// Mitsubishi GX Works2 project: ラダー図整理160913   PLC: Q03UDV

PROGRAM P1
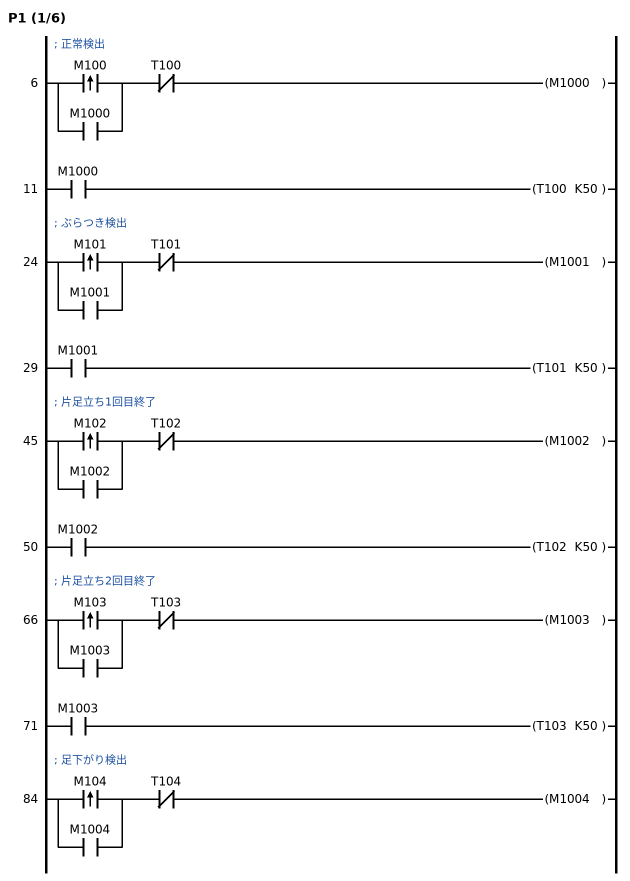
; 正常検出
6     LDP     M100
      OR      M1000
      ANI     T100
      OUT     M1000
11    LD      M1000
      OUT     T100 K50
; ぶらつき検出
24    LDP     M101
      OR      M1001
      ANI     T101
      OUT     M1001
29    LD      M1001
      OUT     T101 K50
; 片足立ち1回目終了
45    LDP     M102
      OR      M1002
      ANI     T102
      OUT     M1002
50    LD      M1002
      OUT     T102 K50
; 片足立ち2回目終了
66    LDP     M103
      OR      M1003
      ANI     T103
      OUT     M1003
71    LD      M1003
      OUT     T103 K50
; 足下がり検出
84    LDP     M104
      OR      M1004
      ANI     T104
      OUT     M1004
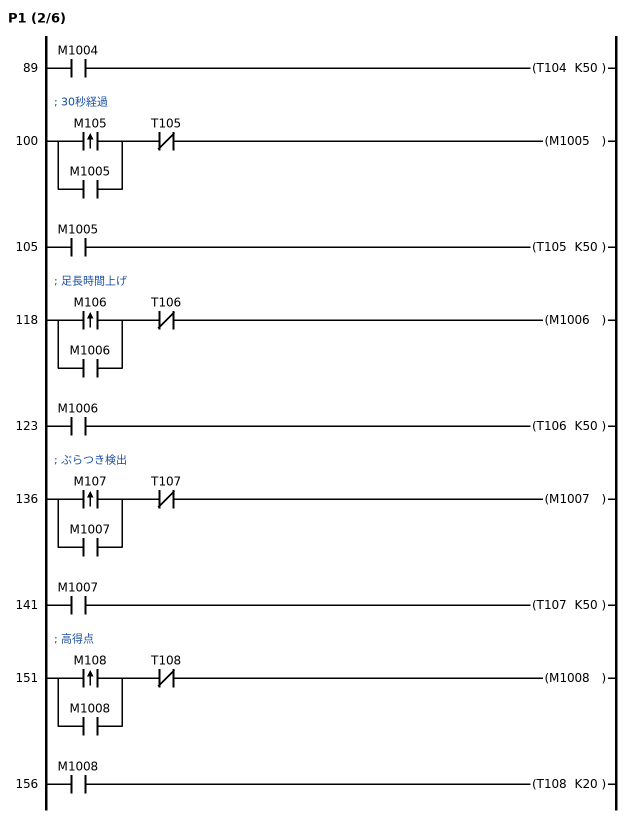
89    LD      M1004
      OUT     T104 K50
; 30秒経過
100   LDP     M105
      OR      M1005
      ANI     T105
      OUT     M1005
105   LD      M1005
      OUT     T105 K50
; 足長時間上げ
118   LDP     M106
      OR      M1006
      ANI     T106
      OUT     M1006
123   LD      M1006
      OUT     T106 K50
; ぶらつき検出
136   LDP     M107
      OR      M1007
      ANI     T107
      OUT     M1007
141   LD      M1007
      OUT     T107 K50
; 高得点
151   LDP     M108
      OR      M1008
      ANI     T108
      OUT     M1008
156   LD      M1008
      OUT     T108 K20
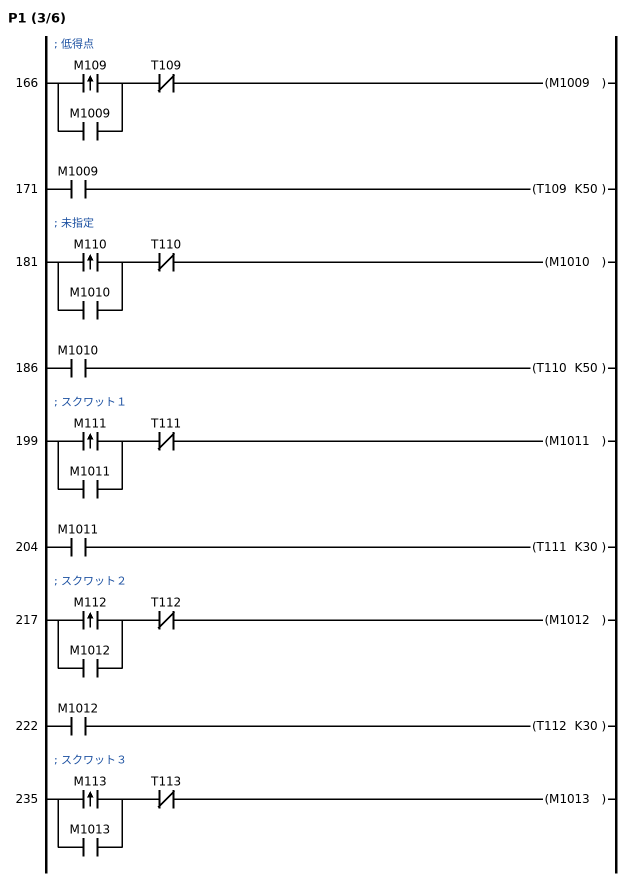
; 低得点
166   LDP     M109
      OR      M1009
      ANI     T109
      OUT     M1009
171   LD      M1009
      OUT     T109 K50
; 未指定
181   LDP     M110
      OR      M1010
      ANI     T110
      OUT     M1010
186   LD      M1010
      OUT     T110 K50
; スクワット１
199   LDP     M111
      OR      M1011
      ANI     T111
      OUT     M1011
204   LD      M1011
      OUT     T111 K30
; スクワット２
217   LDP     M112
      OR      M1012
      ANI     T112
      OUT     M1012
222   LD      M1012
      OUT     T112 K30
; スクワット３
235   LDP     M113
      OR      M1013
      ANI     T113
      OUT     M1013
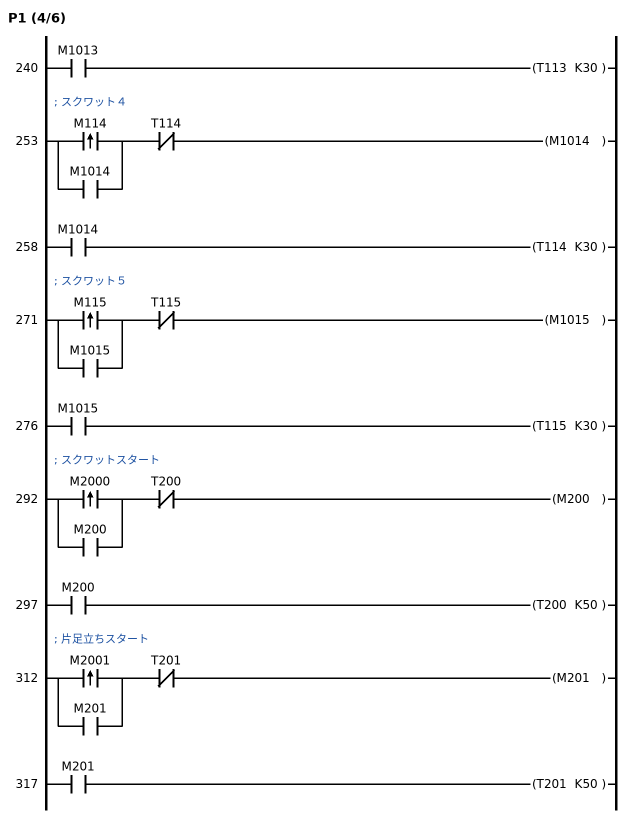
240   LD      M1013
      OUT     T113 K30
; スクワット４
253   LDP     M114
      OR      M1014
      ANI     T114
      OUT     M1014
258   LD      M1014
      OUT     T114 K30
; スクワット５
271   LDP     M115
      OR      M1015
      ANI     T115
      OUT     M1015
276   LD      M1015
      OUT     T115 K30
; スクワットスタート
292   LDP     M2000
      OR      M200
      ANI     T200
      OUT     M200
297   LD      M200
      OUT     T200 K50
; 片足立ちスタート
312   LDP     M2001
      OR      M201
      ANI     T201
      OUT     M201
317   LD      M201
      OUT     T201 K50
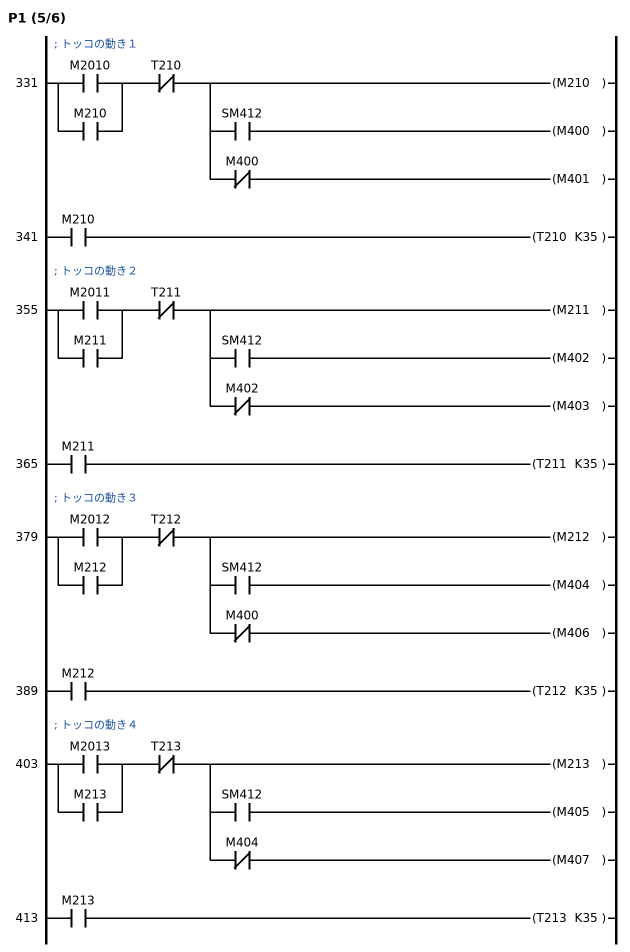
; トッコの動き１
331   LD      M2010
      OR      M210
      ANI     T210
      OUT     M210
      MPS
      AND     SM412
      OUT     M400
      MPP
      ANI     M400
      OUT     M401
341   LD      M210
      OUT     T210 K35
; トッコの動き２
355   LD      M2011
      OR      M211
      ANI     T211
      OUT     M211
      MPS
      AND     SM412
      OUT     M402
      MPP
      ANI     M402
      OUT     M403
365   LD      M211
      OUT     T211 K35
; トッコの動き３
379   LD      M2012
      OR      M212
      ANI     T212
      OUT     M212
      MPS
      AND     SM412
      OUT     M404
      MPP
      ANI     M400
      OUT     M406
389   LD      M212
      OUT     T212 K35
; トッコの動き４
403   LD      M2013
      OR      M213
      ANI     T213
      OUT     M213
      MPS
      AND     SM412
      OUT     M405
      MPP
      ANI     M404
      OUT     M407
413   LD      M213
      OUT     T213 K35
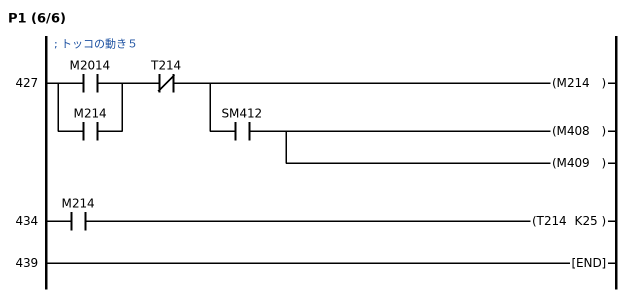
; トッコの動き５
427   LD      M2014
      OR      M214
      ANI     T214
      OUT     M214
      AND     SM412
      OUT     M408
      OUT     M409
434   LD      M214
      OUT     T214 K25
439   END
END_PROGRAM

PROGRAM P2
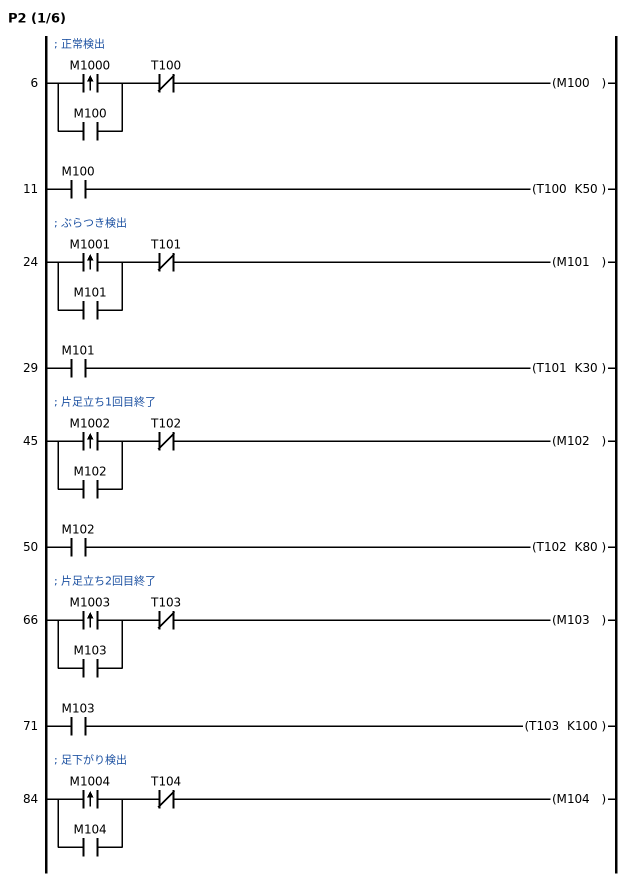
; 正常検出
6     LDP     M1000
      OR      M100
      ANI     T100
      OUT     M100
11    LD      M100
      OUT     T100 K50
; ぶらつき検出
24    LDP     M1001
      OR      M101
      ANI     T101
      OUT     M101
29    LD      M101
      OUT     T101 K30
; 片足立ち1回目終了
45    LDP     M1002
      OR      M102
      ANI     T102
      OUT     M102
50    LD      M102
      OUT     T102 K80
; 片足立ち2回目終了
66    LDP     M1003
      OR      M103
      ANI     T103
      OUT     M103
71    LD      M103
      OUT     T103 K100
; 足下がり検出
84    LDP     M1004
      OR      M104
      ANI     T104
      OUT     M104
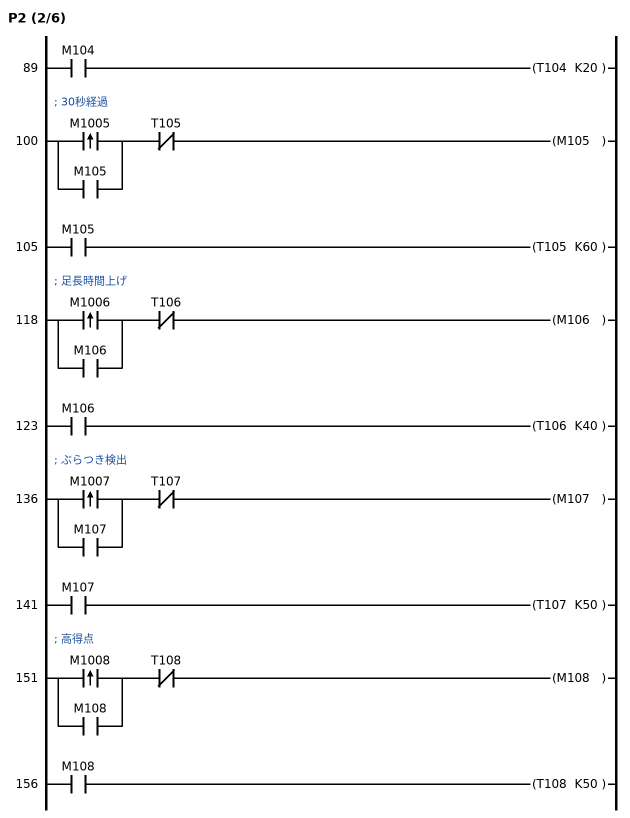
89    LD      M104
      OUT     T104 K20
; 30秒経過
100   LDP     M1005
      OR      M105
      ANI     T105
      OUT     M105
105   LD      M105
      OUT     T105 K60
; 足長時間上げ
118   LDP     M1006
      OR      M106
      ANI     T106
      OUT     M106
123   LD      M106
      OUT     T106 K40
; ぶらつき検出
136   LDP     M1007
      OR      M107
      ANI     T107
      OUT     M107
141   LD      M107
      OUT     T107 K50
; 高得点
151   LDP     M1008
      OR      M108
      ANI     T108
      OUT     M108
156   LD      M108
      OUT     T108 K50
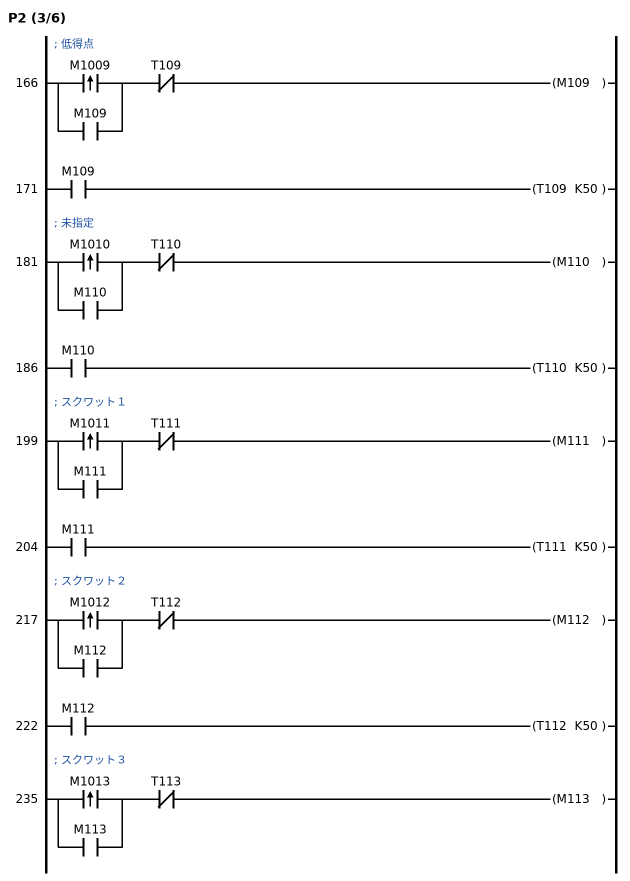
; 低得点
166   LDP     M1009
      OR      M109
      ANI     T109
      OUT     M109
171   LD      M109
      OUT     T109 K50
; 未指定
181   LDP     M1010
      OR      M110
      ANI     T110
      OUT     M110
186   LD      M110
      OUT     T110 K50
; スクワット１
199   LDP     M1011
      OR      M111
      ANI     T111
      OUT     M111
204   LD      M111
      OUT     T111 K50
; スクワット２
217   LDP     M1012
      OR      M112
      ANI     T112
      OUT     M112
222   LD      M112
      OUT     T112 K50
; スクワット３
235   LDP     M1013
      OR      M113
      ANI     T113
      OUT     M113
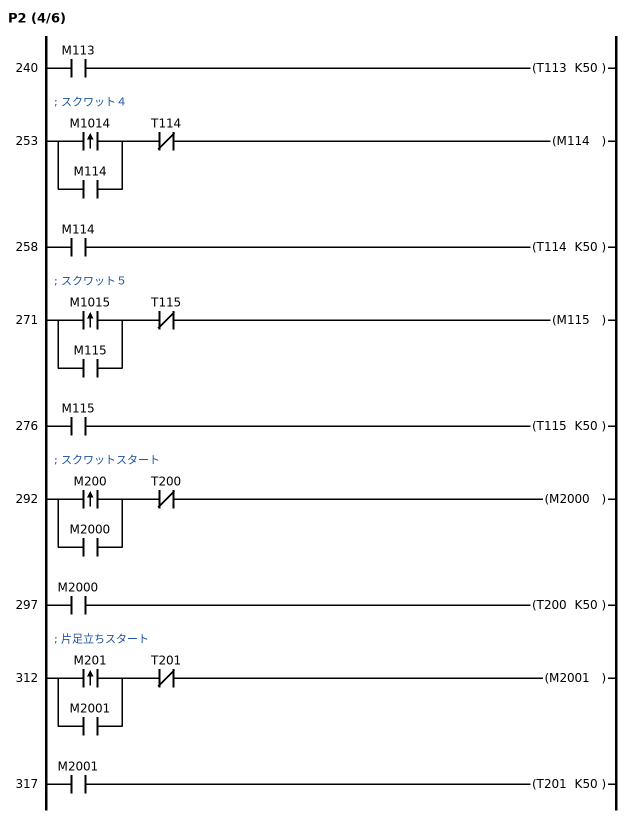
240   LD      M113
      OUT     T113 K50
; スクワット４
253   LDP     M1014
      OR      M114
      ANI     T114
      OUT     M114
258   LD      M114
      OUT     T114 K50
; スクワット５
271   LDP     M1015
      OR      M115
      ANI     T115
      OUT     M115
276   LD      M115
      OUT     T115 K50
; スクワットスタート
292   LDP     M200
      OR      M2000
      ANI     T200
      OUT     M2000
297   LD      M2000
      OUT     T200 K50
; 片足立ちスタート
312   LDP     M201
      OR      M2001
      ANI     T201
      OUT     M2001
317   LD      M2001
      OUT     T201 K50
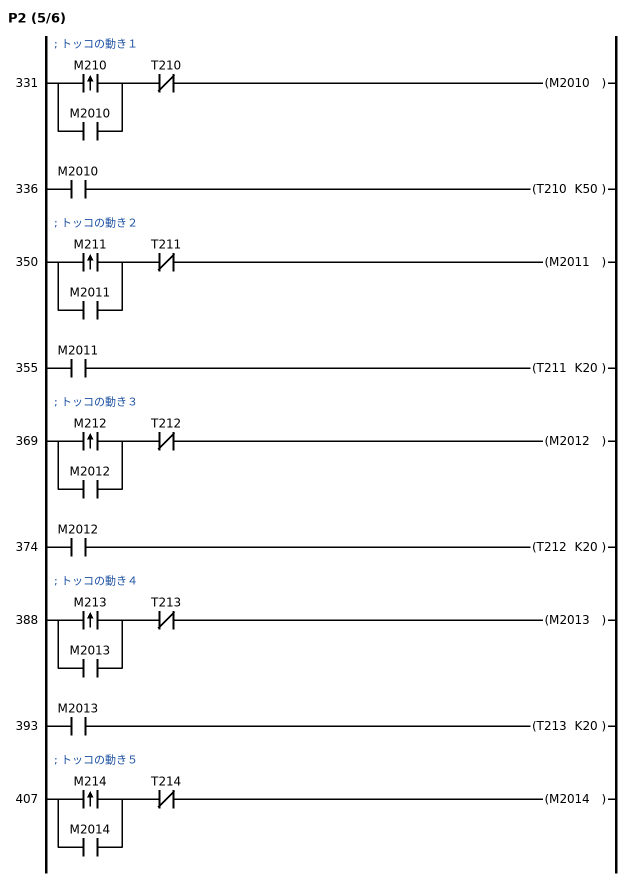
; トッコの動き１
331   LDP     M210
      OR      M2010
      ANI     T210
      OUT     M2010
336   LD      M2010
      OUT     T210 K50
; トッコの動き２
350   LDP     M211
      OR      M2011
      ANI     T211
      OUT     M2011
355   LD      M2011
      OUT     T211 K20
; トッコの動き３
369   LDP     M212
      OR      M2012
      ANI     T212
      OUT     M2012
374   LD      M2012
      OUT     T212 K20
; トッコの動き４
388   LDP     M213
      OR      M2013
      ANI     T213
      OUT     M2013
393   LD      M2013
      OUT     T213 K20
; トッコの動き５
407   LDP     M214
      OR      M2014
      ANI     T214
      OUT     M2014
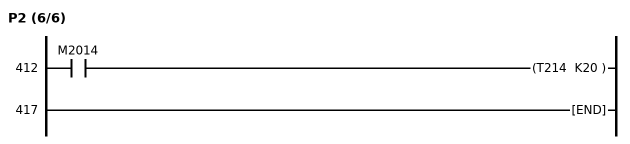
412   LD      M2014
      OUT     T214 K20
417   END
END_PROGRAM
